# EPICS autosave request: dxpApp/Db/dxpSCA_settings.req
$(P)$(R)SCA$(N)Low
$(P)$(R)SCA$(N)High
